{attribute 'GeneratedUsingTerminal: EK1122-0000-0018'}
{attribute addProperty BoxType "EK1122-0000-0018"}
{attribute addProperty Id "Term_187_EK1100Term_187_EK1100_648C31BD62Term_207_EK1100Term_207_EK1100_2D36550A62"}
{attribute addProperty CRC "1976016210"}
{attribute addProperty Size "124"}
{attribute addProperty Name "Term 186 (EK1122)"}
TYPE Term_186_EK1122_75C79D52 EXTENDS EK1122_1FC0878B :
STRUCT
	{attribute addProperty Name "Term 187 (EK1100)"}
	{attribute addProperty PreviousPort "Term 186 (EK1122) : D"}
	{attribute addProperty SyncUnit "default"}
	Term_187_EK1100 : Term_187_EK1100_648C31BD;
	{attribute addProperty Name "Term 207 (EK1100)"}
	{attribute addProperty PreviousPort "Term 186 (EK1122) : B"}
	{attribute addProperty SyncUnit "default"}
	Term_207_EK1100 : Term_207_EK1100_2D36550A;
END_STRUCT
END_TYPE

(* stored: Version 1.2.0.0, ProductVersion 3.1.4024.11
   DUT Term_186_EK1122_75C79D52: Id {527bcac9-5902-0cba-0591-2b6c6f0f55ad} *)
